// Block: PPrgArchive16

DATA_BLOCK PPrgArchive16
VERSION : 0.1
   NON_RETAIN
   VAR
      PRG : Array[1501..1600] of PPrg_Data;
   END_VAR

BEGIN
   // No initialization required
END_DATA_BLOCK
